// TIA Portal project "babu_microwave" (V15)

(* hardware
DEVICE "S7-1200 station_1"  S7-1200 Station
   slot 0: "Rack_0"  S7-1200 Rack  Rack  V1.0
   slot 1: "PLC_1"  CPU 1212C DC/DC/DC  6ES7 212-1AE40-0XB0  V4.2
*)

// ===== PLC "PLC_1"  CPU 1212C DC/DC/DC =====

VAR_GLOBAL   // PLC tag table "Default tag table"
   "Food Tray" AT %M0.0 : Bool;
   "Microwave Wait" AT %M0.3 : Bool;
   "PreHeat" AT %Q0.1 : Bool;
   "Maintain Temperature" AT %M0.5 : Bool;
   "Cool Down" AT %Q0.2 : Bool;
END_VAR

VAR_GLOBAL   // PLC tag table "Tag table_1"
   "Microwave Heat" AT %Q0.0 : Bool;
   "Microwave Heat Memory State" AT %M0.1 : Bool;
   "Microwave Heat Memory" AT %M0.2 : Bool;
   "Alarm" AT %Q0.3 : Bool;
   "Alarm Memory" AT %M0.4 : Bool;
   "Microwave Cool" AT %Q0.5 : Bool;
   "Push Button" AT %M0.6 : Bool;
   "MEMORY BIT FOR OWEN" AT %M0.7 : Bool;
END_VAR

// folder: System blocks/Program resources

DATA_BLOCK "IEC_Timer_0_DB"   // DB1
{ S7_Optimized_Access := 'TRUE' }
AUTHOR : Simatic
FAMILY : IEC
NAME : IEC_TMR
VERSION : 1.0
// stored: InstanceOfName IEC_TIMER
"IEC_TIMER"
BEGIN
END_DATA_BLOCK

DATA_BLOCK "IEC_Timer_0_DB_2"   // DB3
{ S7_Optimized_Access := 'TRUE' }
AUTHOR : Simatic
FAMILY : IEC
NAME : IEC_TMR
VERSION : 1.0
// stored: InstanceOfName IEC_TIMER
"IEC_TIMER"
BEGIN
END_DATA_BLOCK

DATA_BLOCK "IEC_Timer_0_DB_3"   // DB4
{ S7_Optimized_Access := 'TRUE' }
AUTHOR : Simatic
FAMILY : IEC
NAME : IEC_TMR
VERSION : 1.0
// stored: InstanceOfName IEC_TIMER
"IEC_TIMER"
BEGIN
END_DATA_BLOCK

// folder: (top level)

ORGANIZATION_BLOCK "Main"   // OB1, LAD, ProgramCycle
TITLE = "Main Program Sweep (Cycle)"
{ S7_Optimized_Access := 'TRUE' }
VERSION : 0.1
   VAR_INPUT
      Initial_Call : Bool;   // Initial call of this OB
      Remanence : Bool;   // =True, if remanent data are available
   END_VAR
   VAR_TEMP   // added for the SCL form of the ladder/FBD networks
      _w1 : Bool;
      _w2 : Bool;
   END_VAR
BEGIN

REGION Network 1
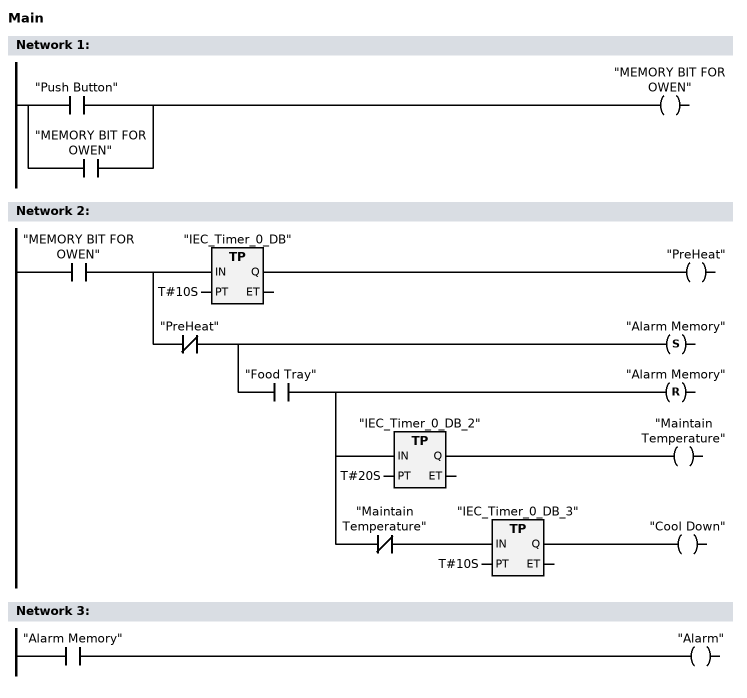
   RUNG wire#powerrail
      Contact( "Push Button" )
      wire#w1
      Coil( "MEMORY BIT FOR OWEN" )
   END_RUNG
   RUNG wire#powerrail
      Contact( "MEMORY BIT FOR OWEN" )
   END_RUNG wire#w1
   // the same network as SCL:
   "MEMORY BIT FOR OWEN" := "Push Button" OR "MEMORY BIT FOR OWEN";
END_REGION

REGION Network 2
   "IEC_Timer_0_DB".TP(IN := "MEMORY BIT FOR OWEN", PT := T#10S);
   "PreHeat" := "IEC_Timer_0_DB".Q;
   #_w1 := "MEMORY BIT FOR OWEN" AND NOT "PreHeat";
   IF #_w1 THEN "Alarm Memory" := TRUE; END_IF;
   #_w2 := #_w1 AND "Food Tray";
   IF #_w2 THEN "Alarm Memory" := FALSE; END_IF;
   "IEC_Timer_0_DB_2".TP(IN := #_w2, PT := T#20S);
   "Maintain Temperature" := "IEC_Timer_0_DB_2".Q;
   "IEC_Timer_0_DB_3".TP(IN := #_w2 AND NOT "Maintain Temperature", PT := T#10S);
   "Cool Down" := "IEC_Timer_0_DB_3".Q;
END_REGION

REGION Network 3
   RUNG wire#powerrail
      Contact( "Alarm Memory" )
      Coil( "Alarm" )
   END_RUNG
   // the same network as SCL:
   "Alarm" := "Alarm Memory";
END_REGION
END_ORGANIZATION_BLOCK